// TIA Portal project "SpeedGate" (V17)

(* hardware
DEVICE "HMI_1"  KTP400 Comfort
   slot 0: "HMI_1"  KTP400 Comfort  6AV2 124-2DC01-0AX0  17.0.0.0
   slot 1: "HMI_RT_1"  KTP400 Comfort  6AV2 124-2DC01-0AX0  17.0.0.0
   slot 5: "HMI_1.IE_CP_1"  PROFINET Interface  17.0.0.0
      slot 1: "PROFINET Interface_1"  PROFINET Interface
         slot 1: "Port_1"  Port
   slot 7: "HMI_1.MPI/DP_CP_1"  MPI/DP Interface  17.0.0.0
DEVICE "S7-1200 station_1"  S7-1200 Station
   slot 0: "Rack_0"  S7-1200 Rack  Rack  V1.0
   slot 1: "PLC_2"  CPU 1211C DC/DC/Rly  6ES7 211-1HE40-0XB0  V4.5
   slot 101: "CM 1241 (RS422/485)_1"  6ES7 241-1CH32-0XB0  V2.2
*)

// ===== PLC "PLC_2"  CPU 1211C DC/DC/Rly =====

VAR_GLOBAL   // PLC tag table "Default tag table"
   "CmdeDroite" AT %I0.0 : Bool;
   "CmdeGauche" AT %I0.1 : Bool;
   "CmdeInitParam" AT %I0.2 : Bool;
   "Tag_5" AT %I1.5 : Bool;
   "Tag_6" AT %I1.4 : Bool;
   "AutoCmde" AT %I0.5 : Bool;
   "ResetAutoCmde" AT %I0.4 : Bool;
   "SensDroite" AT %Q0.0 : Bool;
   "SensGauche" AT %Q0.1 : Bool;
   "InitParam" AT %Q0.2 : Bool;
   "ImageCmdeDroite" AT %M10.0 : Bool;
   "ImageCmdeGauche" AT %M10.1 : Bool;
   "ImageSensDroite" AT %M20.0 : Bool;
   "ImageSensGauche" AT %M20.1 : Bool;
   "MemoSensDroite" AT %M20.2 : Bool;
   "MemoSensGauche" AT %M20.3 : Bool;
   "IHM_SensDroite" AT %M20.4 : Bool;
   "IHM_SensGauche" AT %M20.5 : Bool;
   "System_Byte" AT %MB1 : Byte;
   "FirstScan" AT %M1.0 : Bool;
   "DiagStatusUpdate" AT %M1.1 : Bool;
   "AlwaysTRUE" AT %M1.2 : Bool;
   "AlwaysFALSE" AT %M1.3 : Bool;
   "Clock_Byte" AT %MB0 : Byte;
   "Clock_10Hz" AT %M0.0 : Bool;
   "Clock_5Hz" AT %M0.1 : Bool;
   "Clock_2.5Hz" AT %M0.2 : Bool;
   "Clock_2Hz" AT %M0.3 : Bool;
   "Clock_1.25Hz" AT %M0.4 : Bool;
   "Clock_1Hz" AT %M0.5 : Bool;
   "Clock_0.625Hz" AT %M0.6 : Bool;
   "Clock_0.5Hz" AT %M0.7 : Bool;
   "IHM_REQ" AT %M20.6 : Bool;
   "BUSY" AT %M20.7 : Bool;
   "Addr_baudRate" AT %MW100 : UInt;
   "Addr_Slave" AT %MW102 : UInt;
   "Addr_Main" AT %MW104 : UInt;
   "getBaudValue" AT %M21.0 : Bool;
   "Tag_1" AT %M30.0 : Bool;
   "getSlaveValue" AT %M21.1 : Bool;
   "Tag_2" AT %M50.0 : Bool;
   "Tag_3" AT %M50.1 : Bool;
   "Tag_4" AT %M50.2 : Bool;
   "IHM_InitParam" AT %M21.2 : Bool;
   "ImageInitParam" AT %M21.3 : Bool;
   "MemoInitParam" AT %M21.4 : Bool;
   "LoopCmdeDroite" AT %M50.3 : Bool;
   "LoopCmdeGauche" AT %M50.4 : Bool;
   "IHM_AutoCmde" AT %M21.5 : Bool;
   "IHM_ResetAutoCmde" AT %M21.6 : Bool;
   "TempoDrote" AT %MD30 : Time;
   "tempoGauche" AT %MD34 : Time;
END_VAR

DATA_BLOCK "DataGet"   // DB5
{ S7_Optimized_Access := 'FALSE' }
VERSION : 0.1
   VAR
      Registre : UInt;
   END_VAR
BEGIN
END_DATA_BLOCK

DATA_BLOCK "ADDR_Registre"   // DB7
{ S7_Optimized_Access := 'FALSE' }
VERSION : 0.1
   VAR
      SppedMotor : UInt := 40907;
   END_VAR
BEGIN
END_DATA_BLOCK

// folder: System blocks/Program resources

DATA_BLOCK "IEC_Timer_0_DB"   // DB1
{ S7_Optimized_Access := 'TRUE' }
AUTHOR : Simatic
FAMILY : IEC
NAME : IEC_TMR
VERSION : 1.0
// stored: InstanceOfName IEC_TIMER
"IEC_TIMER"
BEGIN
END_DATA_BLOCK

DATA_BLOCK "IEC_Timer_0_DB_1"   // DB2
{ S7_Optimized_Access := 'TRUE' }
AUTHOR : Simatic
FAMILY : IEC
NAME : IEC_TMR
VERSION : 1.0
// stored: InstanceOfName IEC_TIMER
"IEC_TIMER"
BEGIN
END_DATA_BLOCK

DATA_BLOCK "IEC_Timer_0_DB_2"   // DB6
{ S7_Optimized_Access := 'TRUE' }
AUTHOR : Simatic
FAMILY : IEC
NAME : IEC_TMR
VERSION : 1.0
// stored: InstanceOfName IEC_TIMER
"IEC_TIMER"
BEGIN
END_DATA_BLOCK

DATA_BLOCK "IEC_Timer_0_DB_3"   // DB8
{ S7_Optimized_Access := 'TRUE' }
AUTHOR : Simatic
FAMILY : IEC
NAME : IEC_TMR
VERSION : 1.0
// stored: InstanceOfName IEC_TIMER
"IEC_TIMER"
BEGIN
END_DATA_BLOCK

DATA_BLOCK "IEC_Timer_0_DB_4"   // DB9
{ S7_Optimized_Access := 'TRUE' }
AUTHOR : Simatic
FAMILY : IEC
NAME : IEC_TMR
VERSION : 1.0
// stored: InstanceOfName IEC_TIMER
"IEC_TIMER"
BEGIN
END_DATA_BLOCK

// folder: (top level)

FUNCTION "ImageInput" : Void   // FC1, LAD
{ S7_Optimized_Access := 'TRUE' }
VERSION : 0.1
BEGIN

REGION Network 1
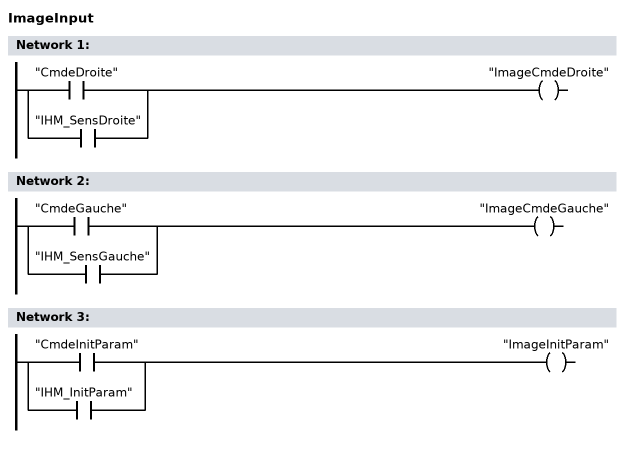
   RUNG wire#powerrail
      Contact( "CmdeDroite" )
      wire#w1
      Coil( "ImageCmdeDroite" )
   END_RUNG
   RUNG wire#powerrail
      Contact( "IHM_SensDroite" )
   END_RUNG wire#w1
   // the same network as SCL:
   "ImageCmdeDroite" := "CmdeDroite" OR "IHM_SensDroite";
END_REGION

REGION Network 2
   RUNG wire#powerrail
      Contact( "CmdeGauche" )
      wire#w1
      Coil( "ImageCmdeGauche" )
   END_RUNG
   RUNG wire#powerrail
      Contact( "IHM_SensGauche" )
   END_RUNG wire#w1
   // the same network as SCL:
   "ImageCmdeGauche" := "CmdeGauche" OR "IHM_SensGauche";
END_REGION

REGION Network 3
   RUNG wire#powerrail
      Contact( "CmdeInitParam" )
      wire#w1
      Coil( "ImageInitParam" )
   END_RUNG
   RUNG wire#powerrail
      Contact( "IHM_InitParam" )
   END_RUNG wire#w1
   // the same network as SCL:
   "ImageInitParam" := "CmdeInitParam" OR "IHM_InitParam";
END_REGION
END_FUNCTION

FUNCTION "CommandeMoteur" : Void   // FC2, LAD
{ S7_Optimized_Access := 'TRUE' }
VERSION : 0.1
BEGIN

REGION Network 1
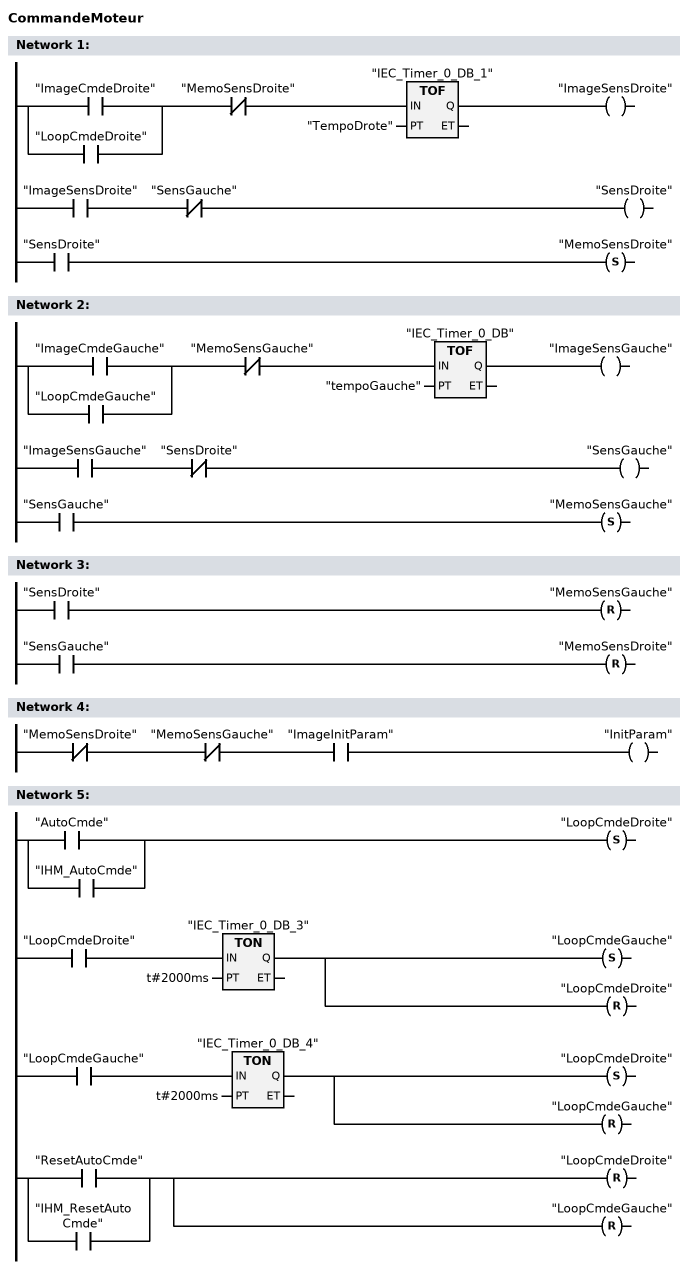
   "IEC_Timer_0_DB_1".TOF(IN := ("ImageCmdeDroite" OR "LoopCmdeDroite") AND NOT "MemoSensDroite",
                          PT := "TempoDrote");
   "ImageSensDroite" := "IEC_Timer_0_DB_1".Q;
   "SensDroite" := "ImageSensDroite" AND NOT "SensGauche";
   IF "SensDroite" THEN "MemoSensDroite" := TRUE; END_IF;
END_REGION

REGION Network 2
   "IEC_Timer_0_DB".TOF(IN := ("ImageCmdeGauche" OR "LoopCmdeGauche") AND NOT "MemoSensGauche",
                        PT := "tempoGauche");
   "ImageSensGauche" := "IEC_Timer_0_DB".Q;
   "SensGauche" := "ImageSensGauche" AND NOT "SensDroite";
   IF "SensGauche" THEN "MemoSensGauche" := TRUE; END_IF;
END_REGION

REGION Network 3
   RUNG wire#powerrail
      Contact( "SensDroite" )
      R_Coil( "MemoSensGauche" )
   END_RUNG
   RUNG wire#powerrail
      Contact( "SensGauche" )
      R_Coil( "MemoSensDroite" )
   END_RUNG
   // the same network as SCL:
   IF "SensDroite" THEN "MemoSensGauche" := FALSE; END_IF;
   IF "SensGauche" THEN "MemoSensDroite" := FALSE; END_IF;
END_REGION

REGION Network 4
   RUNG wire#powerrail
      I_Contact( "MemoSensDroite" )
      I_Contact( "MemoSensGauche" )
      Contact( "ImageInitParam" )
      Coil( "InitParam" )
   END_RUNG
   // the same network as SCL:
   "InitParam" := NOT "MemoSensDroite" AND NOT "MemoSensGauche" AND "ImageInitParam";
END_REGION

REGION Network 5
   IF "AutoCmde" OR "IHM_AutoCmde" THEN "LoopCmdeDroite" := TRUE; END_IF;
   "IEC_Timer_0_DB_3".TON(IN := "LoopCmdeDroite", PT := t#2000ms);
   IF "IEC_Timer_0_DB_3".Q THEN
       "LoopCmdeGauche" := TRUE;
       "LoopCmdeDroite" := FALSE;
   END_IF;
   "IEC_Timer_0_DB_4".TON(IN := "LoopCmdeGauche", PT := t#2000ms);
   IF "IEC_Timer_0_DB_4".Q THEN
       "LoopCmdeDroite" := TRUE;
       "LoopCmdeGauche" := FALSE;
   END_IF;
   IF "ResetAutoCmde" OR "IHM_ResetAutoCmde" THEN
       "LoopCmdeDroite" := FALSE;
       "LoopCmdeGauche" := FALSE;
   END_IF;
END_REGION
END_FUNCTION

FUNCTION "COM_RS485" : Void   // FC3, LAD
{ S7_Optimized_Access := 'TRUE' }
VERSION : 0.1
BEGIN

REGION Network 1
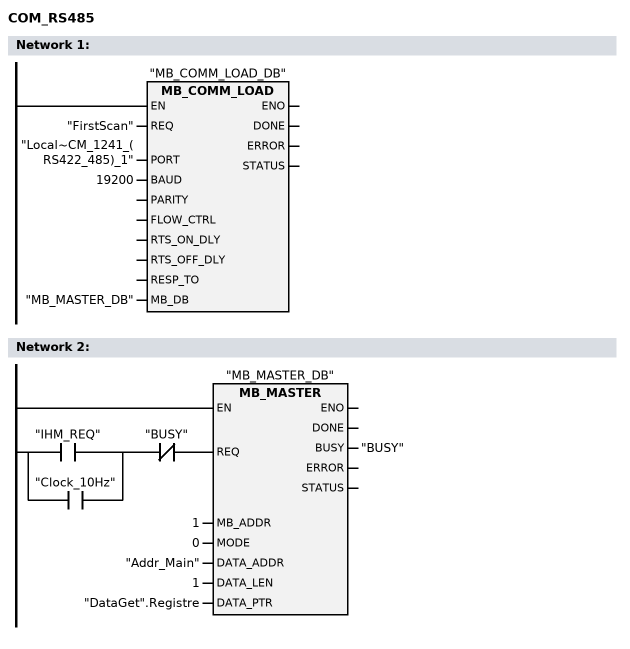
   "MB_COMM_LOAD_DB"(REQ := "FirstScan",   // MB_COMM_LOAD
                     PORT := "Local~CM_1241_(RS422_485)_1",
                     BAUD := 19200,
                     MB_DB := "MB_MASTER_DB");
END_REGION

REGION Network 2
   "MB_MASTER_DB"(REQ := ("IHM_REQ" OR "Clock_10Hz") AND NOT "BUSY",   // MB_MASTER
                  MB_ADDR := 1,
                  MODE := 0,
                  DATA_ADDR := "Addr_Main",
                  DATA_LEN := 1,
                  DATA_PTR := "DataGet".Registre,
                  BUSY => "BUSY");
END_REGION
END_FUNCTION

FUNCTION "ImageRegistre" : Void   // FC4, LAD
{ S7_Optimized_Access := 'TRUE' }
VERSION : 0.1
   VAR_TEMP   // added for the SCL form of the ladder/FBD networks
      _w1 : Bool;
      _w2 : Bool;
   END_VAR
BEGIN

REGION Network 1
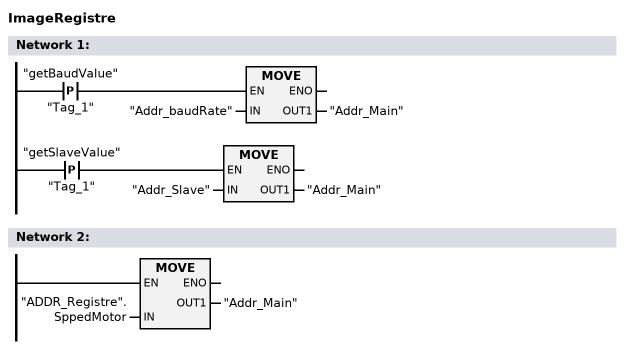
   RUNG wire#powerrail
      P_Contact(operand := "getBaudValue", bit := "Tag_1")
      { S7_GenerateENO := "TRUE" } Move(in := "Addr_baudRate", out1 => "Addr_Main")
   END_RUNG
   RUNG wire#powerrail
      P_Contact(operand := "getSlaveValue", bit := "Tag_1")
      { S7_GenerateENO := "TRUE" } Move(in := "Addr_Slave", out1 => "Addr_Main")
   END_RUNG
   // the same network as SCL:
   #_w1 := "getBaudValue" AND NOT "Tag_1";   // rising edge of "getBaudValue"
   "Tag_1" := "getBaudValue";
   IF #_w1 THEN "Addr_Main" := "Addr_baudRate"; END_IF;
   #_w2 := "getSlaveValue" AND NOT "Tag_1";   // rising edge of "getSlaveValue"
   "Tag_1" := "getSlaveValue";
   IF #_w2 THEN "Addr_Main" := "Addr_Slave"; END_IF;
END_REGION

REGION Network 2
   RUNG wire#powerrail
      { S7_GenerateENO := "TRUE" } Move(in := "ADDR_Registre".SppedMotor, out1 => "Addr_Main")
   END_RUNG
   // the same network as SCL:
   "Addr_Main" := "ADDR_Registre".SppedMotor;
END_REGION
END_FUNCTION

FUNCTION "commandeMoteurRS485" : Void   // FC5, LAD
{ S7_Optimized_Access := 'TRUE' }
VERSION : 0.1
BEGIN

REGION Network 1
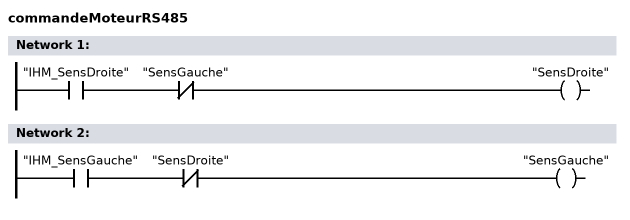
   RUNG wire#powerrail
      Contact( "IHM_SensDroite" )
      I_Contact( "SensGauche" )
      Coil( "SensDroite" )
   END_RUNG
   // the same network as SCL:
   "SensDroite" := "IHM_SensDroite" AND NOT "SensGauche";
END_REGION

REGION Network 2
   RUNG wire#powerrail
      Contact( "IHM_SensGauche" )
      I_Contact( "SensDroite" )
      Coil( "SensGauche" )
   END_RUNG
   // the same network as SCL:
   "SensGauche" := "IHM_SensGauche" AND NOT "SensDroite";
END_REGION
END_FUNCTION

ORGANIZATION_BLOCK "Main"   // OB1, LAD, ProgramCycle
{ S7_Optimized_Access := 'TRUE' }
VERSION : 0.1
BEGIN

REGION Network 1
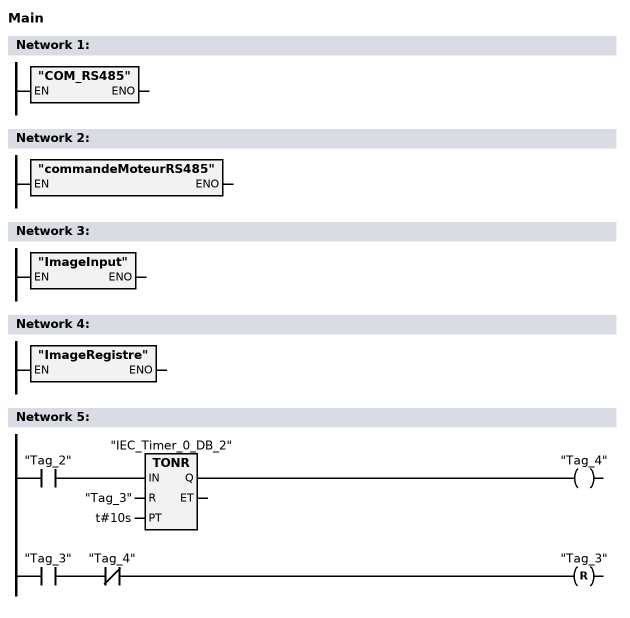
   RUNG wire#powerrail
      "COM_RS485"()
   END_RUNG
   // the same network as SCL:
   "COM_RS485"();
END_REGION

REGION Network 2
   RUNG wire#powerrail
      "commandeMoteurRS485"()
   END_RUNG
   // the same network as SCL:
   "commandeMoteurRS485"();
END_REGION

REGION Network 3
   RUNG wire#powerrail
      "ImageInput"()
   END_RUNG
   // the same network as SCL:
   "ImageInput"();
END_REGION

REGION Network 4
   RUNG wire#powerrail
      "ImageRegistre"()
   END_RUNG
   // the same network as SCL:
   "ImageRegistre"();
END_REGION

REGION Network 5
   "IEC_Timer_0_DB_2".TONR(IN := "Tag_2", R := "Tag_3", PT := t#10s);
   "Tag_4" := "IEC_Timer_0_DB_2".Q;
   IF "Tag_3" AND NOT "Tag_4" THEN "Tag_3" := FALSE; END_IF;
END_REGION
END_ORGANIZATION_BLOCK

(* ===== HMI "HMI_RT_1" =====
system functions are stored by id; their names below are inferred from use
connection "HMI_Connection_2": ETHERNET, S7_1200_OMS

HMI tags "Default tag table"
   "IHM_SensDroite" : Bool = PLC IHM_SensDroite AT %M20.4, 1 s
   "IHM_SensGauche" : Bool = PLC IHM_SensGauche AT %M20.5, 1 s
   "IHM_InitParam" : Bool = PLC IHM_InitParam AT %M21.2, 1 s
   "IHM_AutoCmde" : Bool = PLC IHM_AutoCmde AT %M21.5, 1 s
   "IHM_ResetAutoCmde" : Bool = PLC IHM_ResetAutoCmde AT %M21.6, 1 s
   "TempoDrote" : Time = PLC TempoDrote AT %MD30, 1 s
   "tempoGauche" : Time = PLC tempoGauche AT %MD34, 1 s

screen "Root screen" 480x272, template "Template_1"
   Button "Button_1" at 17,20 size 96x32; TextOff 'DROITE'
      on Press: SetBit("IHM_SensDroite")
      on Release: ResetBit("IHM_SensDroite")
   Button "Button_2" at 276,20 size 96x32; TextOff 'GAUCHE'
      on Press: SetBit("IHM_SensGauche")
      on Release: ResetBit("IHM_SensGauche")
   Button "Button_3" at 143,126 size 96x32; TextOff 'INIT PARAM'
      on Press: SetBit("IHM_InitParam")
      on Release: ResetBit("IHM_InitParam")
   Button "Button_4" at 17,210 size 96x32; TextOff 'AUTO MODE'
      on Press: SetBit("IHM_AutoCmde")
      on Release: ResetBit("IHM_AutoCmde")
   Button "Button_5" at 276,209 size 96x32; TextOff 'RESET MODE'
      on Press: SetBit("IHM_ResetAutoCmde")
      on Release: ResetBit("IHM_ResetAutoCmde")
   IOField "I/O field_1" at 22,68 size 96x32; FormatPattern s9999999999
      ProcessValue <- "TempoDrote"
   IOField "I/O field_2" at 276,68 size 96x32; FormatPattern s9999999999
      ProcessValue <- "tempoGauche"

Template "Template_1" 480x272
   Button "Start screen" at 415,1 size 63x63; TextOff 'Start screen'; PictureOff "NavigateHome_KTP400_Comfort_TR"; PictureOn "NavigateHome_KTP400_Comfort_TR"
      on Release: ActivateScreen("Root screen", 0)
   Button "Template_Button" at 415,70 size 63x63; TextOff 'Text'
   Button "Template_Button_1" at 415,138 size 63x63; TextOff 'Text'
   Button "Exit" at 415,207 size 63x63; TextOff 'Exit'; PictureOff "ExitRuntime_KTP400_Comfort_TR"; PictureOn "ExitRuntime_KTP400_Comfort_TR"
      on Release: StopRuntime(0)
*)